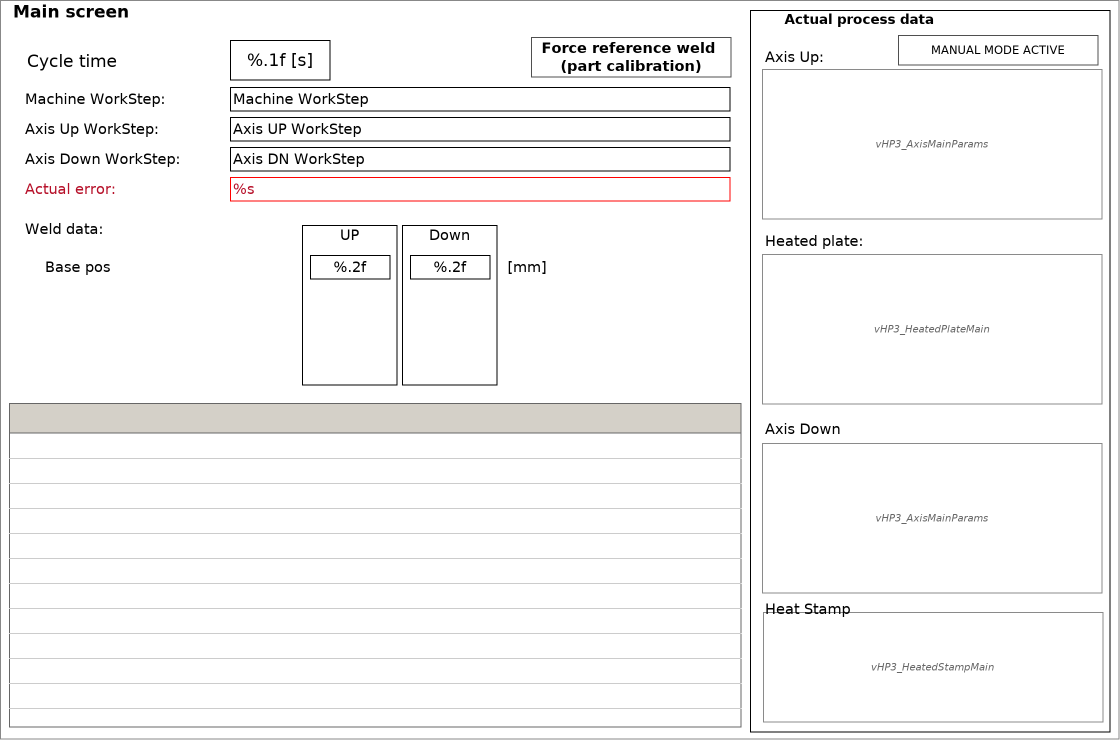
VISUALIZATION vHP3_MachineSub_Main  // 1120x740
VAR_IN_OUT
	fbHP: fbHPv3_Control;
END_VAR
    RoundedRectangle (10,0 300x26), "Main screen"
    Table (9,403 732x324), data array: fbHP.fbTimeStats.astTT
        p3854506369: fbHP.fbTimeStats.astTT[INDEX].sStepName
        p1892666644: fbHP.fbTimeStats.astTT[INDEX].rStepTime
        p2232123230: Step name
        p511219082: Step time
        p1128707560: fbHP.fbTimeStats.uiTTLastIndex
    Label (42,255 260x24), "Base pos"
    RoundedRectangle (402,225 95x160), "Down"
    RoundedRectangle (302,225 95x160), "UP"
    Rectangle (310,255 80x24), "%.2f", text variable: fbHP.fbAxisUp.lrBasePos_mm
    Label (502,255 50x24), "[mm]"
    Rectangle (410,255 80x24), "%.2f", text variable: fbHP.fbAxisDn.lrBasePos_mm
    Label (22,87 200x24), "Machine WorkStep:"
    Label (22,117 200x24), "Axis Up WorkStep:"
    Label (22,147 200x24), "Axis Down WorkStep:"
    Rectangle (230,87 500x24), "Machine WorkStep", text list: 'tlHPv3', text index: fbHP.iHMI_StepName
    Rectangle (230,117 500x24), "Axis UP WorkStep", text list: 'tlHPv3', text index: fbHP.fbAxisUp.iHMI_StepName
    Rectangle (230,147 500x24), "Axis DN WorkStep", text list: 'tlHPv3', text index: fbHP.fbAxisDn.iHMI_StepName
    Rectangle (230,40 100x40), "%.1f [s]", text variable: TIME_TO_REAL(fbHP.fbTON_OperationTime.ET)/1000
    Label (24,41 204x40), "Cycle time"
    RoundedRectangle (750,10 360x722), "Actual process data"
    Label (762,45 200x24), "Axis Up:"
    Frame (762,69 340x150)
        shows vHP3_AxisMainParams(fbAxis := fbHP.fbAxisUp)
    Label (762,417 200x24), "Axis Down"
    Frame (762,443 340x150)
        shows vHP3_AxisMainParams(fbAxis := fbHP.fbAxisDn)
    Label (762,229 200x24), "Heated plate:"
    Frame (762,254 340x150)
        shows vHP3_HeatedPlateMain(fbHP := fbHP)
    Rectangle (898,35 200x30), "MANUAL MODE ACTIVE", invisible if: NOT fbHP.bManualMode
    Label (22,217 200x24), "Weld data:"
    Rectangle (531,37 200x40), "Force reference weld (part calibration)", colour toggle: fbHP.bAxisPartCalibtarion, input disabled if: fbHP.iWorkStep > 10
        OnMouseDown: execute {
            fbHP.fbAxisUp.IsCalibrated := FALSE;
            fbHP.fbAxisDn.IsCalibrated := FALSE;
            fbHP.bAxisPartCalibtarion := TRUE;
        }
    Label (22,177 200x24), "Actual error:", invisible if: fbHP.iWorkStep <90
    Rectangle (230,177 500x24), "%s", text variable: TO_STRING(fbHP.nError), invisible if: fbHP.iWorkStep <90
    Frame (763,612 340x110), invisible if: Not fbHP.bMarkingAsembled
        shows vHP3_HeatedStampMain(fbHP := fbHP)
    Label (762,597 200x24), "Heat Stamp", invisible if: Not fbHP.bMarkingAsembled
END_VISUALIZATION

(* stored: Version 1.1.0.1, ProductVersion 3.1.4024.13
   Visu vHP3_MachineSub_Main: Id {ad33e5d7-4b7c-4021-9e02-6a52288ded3a} *)
